% RSLogix 500 project ML1500_BAK025.RSS, saved by version 10.00.00.00 %
PROJECT "ML1500"    % processor: MicroLogix 1500; MAIN_PROG %

PROGRAM FILES
  LAD 2 "MAIN_PROG"  24 rungs

DATA FILES
  O0 OUTPUT  6 elements
  I1 INPUT  18 elements
  S2 STATUS  66 elements
  B3 BINARY  2 elements
  T4 TIMER  5 elements
  C5 COUNTER  1 elements
  R6 CONTROL  1 elements
  N7 INTEGER  1 elements
  F8 FLOAT  1 elements

LADDER 2 "MAIN_PROG"
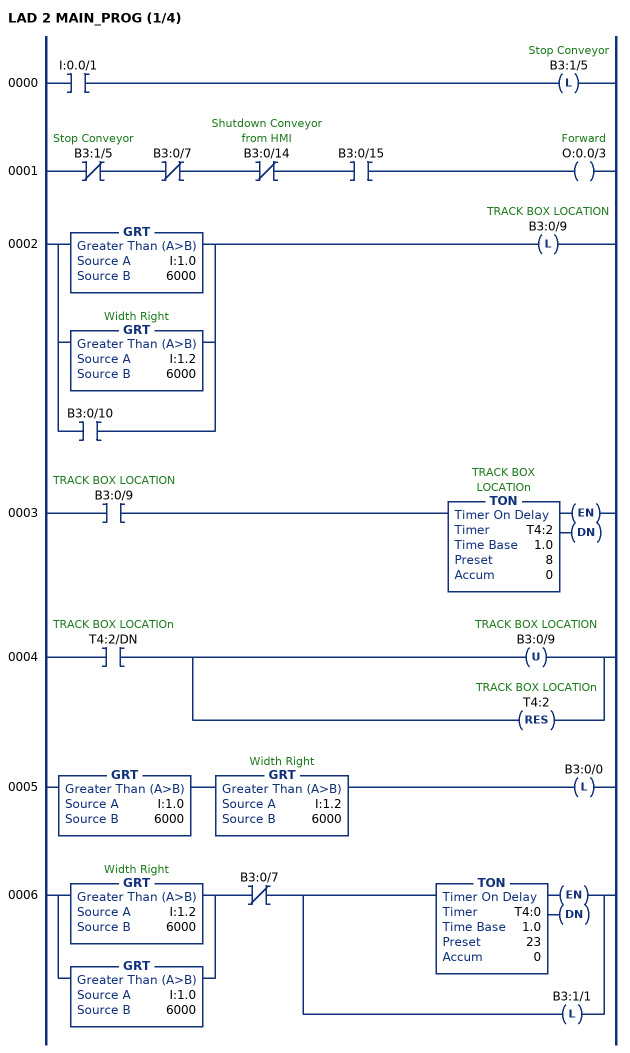
% Rung: 0 %
SOR XIC I:0.0/1 OTL B3:1/5 EOR
%   B3:1/5  "Stop Conveyor" %
% Rung: 1 %
SOR XIO B3:1/5 XIO B3:0/7 XIO B3:0/14 XIC B3:0/15 OTE O:0.0/3 EOR
%   B3:1/5  "Stop Conveyor" %
%   B3:0/14  "Shutdown Conveyor from HMI" %
%   O:0.0/3  "Forward" %
% Rung: 2 %
SOR BST GRT I:1.0 6000 NXB BST GRT I:1.2 6000 NXB XIC B3:0/10 BND BND OTL B3:0/9 EOR
%   I:1.2  "Width Right" %
%   B3:0/9  "TRACK BOX LOCATION" %
% Rung: 3 %
SOR XIC B3:0/9 TON T4:2 1.0 8 0 EOR
%   B3:0/9  "TRACK BOX LOCATION" %
%   T4:2  "TRACK BOX LOCATIOn" %
% Rung: 4 %
SOR XIC T4:2/DN BST OTU B3:0/9 NXB RES T4:2 BND EOR
%   T4:2  "TRACK BOX LOCATIOn" %
%   B3:0/9  "TRACK BOX LOCATION" %
% Rung: 5 %
SOR GRT I:1.0 6000 GRT I:1.2 6000 OTL B3:0/0 EOR
%   I:1.2  "Width Right" %
% Rung: 6 %
SOR BST GRT I:1.2 6000 NXB GRT I:1.0 6000 BND XIO B3:0/7 BST TON T4:0 1.0 23 0 NXB OTL B3:1/1 BND EOR
%   I:1.2  "Width Right" %

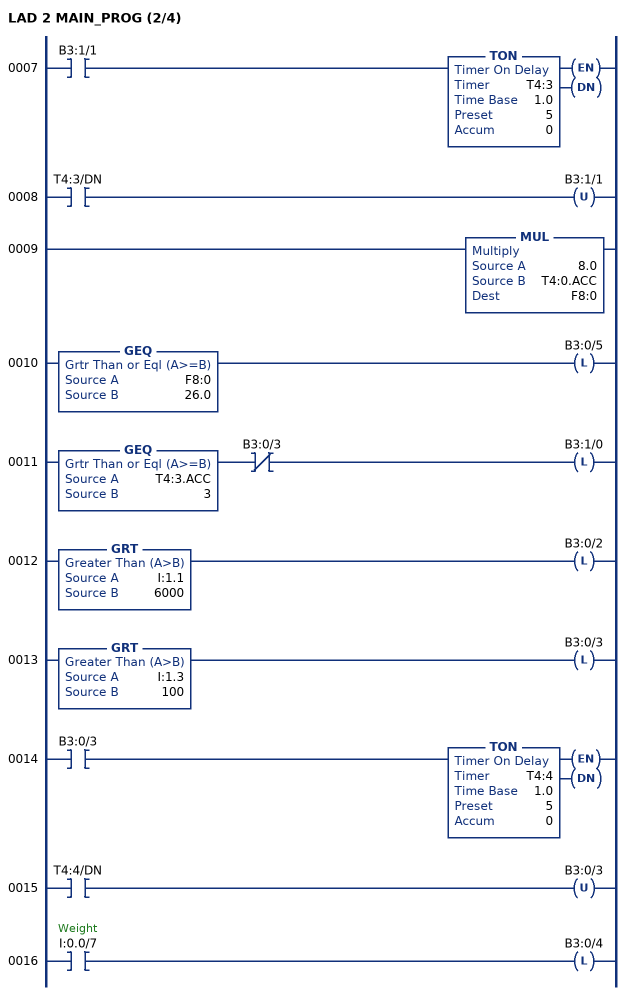
% Rung: 7 %
SOR XIC B3:1/1 TON T4:3 1.0 5 0 EOR
% Rung: 8 %
SOR XIC T4:3/DN OTU B3:1/1 EOR
% Rung: 9 %
SOR MUL 8.0 T4:0.ACC F8:0 EOR
% Rung: 10 %
SOR GEQ F8:0 26.0 OTL B3:0/5 EOR
% Rung: 11 %
SOR GEQ T4:3.ACC 3 XIO B3:0/3 OTL B3:1/0 EOR
% Rung: 12 %
SOR GRT I:1.1 6000 OTL B3:0/2 EOR
% Rung: 13 %
SOR GRT I:1.3 100 OTL B3:0/3 EOR
% Rung: 14 %
SOR XIC B3:0/3 TON T4:4 1.0 5 0 EOR
% Rung: 15 %
SOR XIC T4:4/DN OTU B3:0/3 EOR
% Rung: 16 %
SOR XIC I:0.0/7 OTL B3:0/4 EOR
%   I:0.0/7  "Weight" %

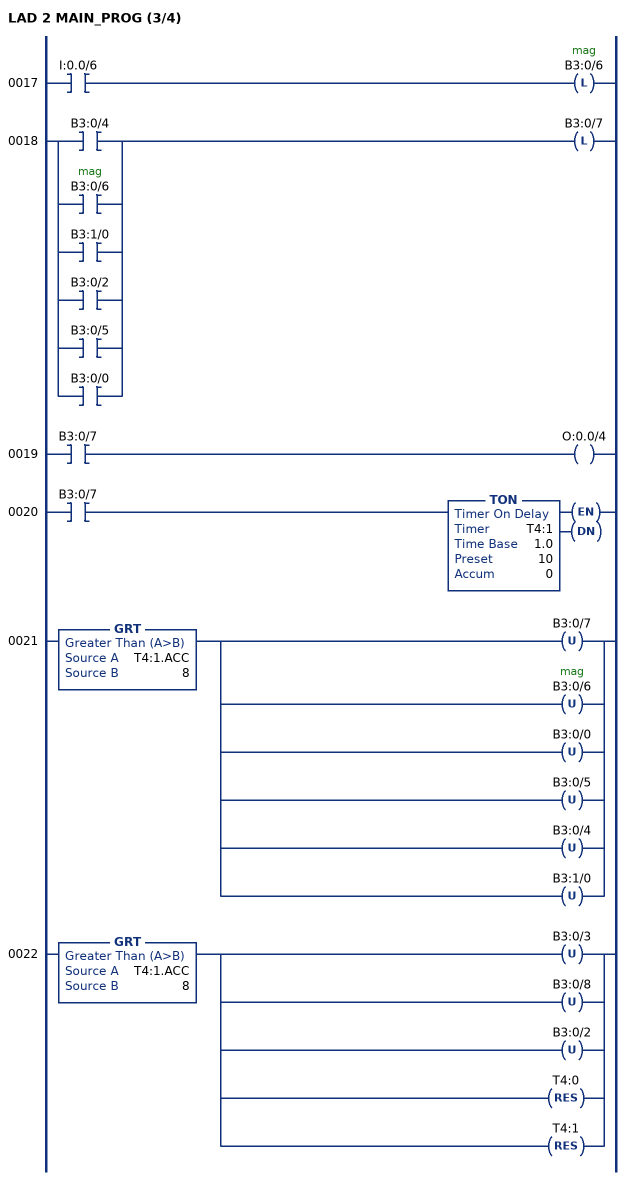
% Rung: 17 %
SOR XIC I:0.0/6 OTL B3:0/6 EOR
%   B3:0/6  "mag" %
% Rung: 18 %
SOR BST BST XIC B3:0/4 NXB XIC B3:0/6 BND NXB BST XIC B3:1/0 NXB BST XIC B3:0/2 NXB BST XIC B3:0/5 NXB XIC B3:0/0 BND BND BND BND OTL B3:0/7 EOR
%   B3:0/6  "mag" %
% Rung: 19 %
SOR XIC B3:0/7 OTE O:0.0/4 EOR
% Rung: 20 %
SOR XIC B3:0/7 TON T4:1 1.0 10 0 EOR
% Rung: 21 %
SOR GRT T4:1.ACC 8 BST BST OTU B3:0/7 NXB OTU B3:0/6 BND NXB BST OTU B3:0/0 NXB BST OTU B3:0/5 NXB BST OTU B3:0/4 NXB OTU B3:1/0 BND BND BND BND EOR
%   B3:0/6  "mag" %
% Rung: 22 %
SOR GRT T4:1.ACC 8 BST OTU B3:0/3 NXB BST OTU B3:0/8 NXB BST OTU B3:0/2 NXB BST RES T4:0 NXB RES T4:1 BND BND BND BND EOR

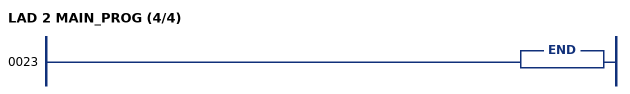
% Rung: 23 %
SOR END EOR

OTHER DOCUMENTED ADDRESSES
  I:0.0/8  "Weight"
  O:0.0/5  "BACKWARD"
  O:0.0/6  "FORWARD"

DATA TABLE (non-zero values as saved)
DATA B3
% B3:0 % 0X8000 0X0020
DATA T4
% .PRE .ACC %
% T4:0 % 23 0
% T4:1 % 10 0
% T4:2 % 8 0
% T4:3 % 5 0
% T4:4 % 5 0
